{attribute 'qualified_only'}
{attribute 'strict'}
TYPE EFeedbackMsgBisL405 :
(
	DataCarrierMsg := 10
);
END_TYPE

(* stored: Version 1.1.0.1, ProductVersion 3.1.4024.12
   DUT EFeedbackMsgBisL405: Id {aa3ba0e1-b093-4871-9d4b-6f1743049d1b} *)
